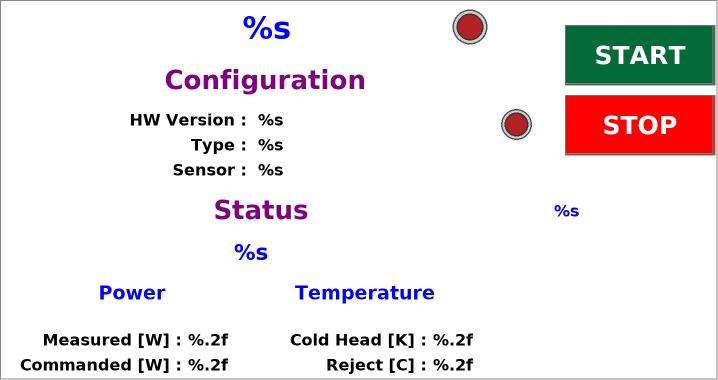
VISUALIZATION GUI_TEMPLATE_CRYOTELGT  // 718x380
VAR_IN_OUT
	m_Instance:	FB_CRYO_CRYOTELGT;
	m_bEnable:	BOOL;	// Flag to start/stop the cooler
END_VAR
    Rectangle (159,65 213x30), "Configuration"
    Rectangle (186,195 150x30), "Status"
    Rectangle (25,325 160x30), "Measured [W] :", tooltip "'P' command: Measured Power"
    Rectangle (185,325 70x30), "%.2f", text variable: m_Instance.stat.lrPowerMeasured
    Rectangle (152,10 230x36), "%s", text variable: m_Instance.in_sName
    Rectangle (255,155 110x30), "%s", text variable: m_Instance.stat.sSensor
    Rectangle (255,105 100x30), "%s", text variable: m_Instance.stat.sVersion
    Rectangle (255,130 100x30), "%s", text variable: m_Instance.stat.sMode
    Button (565,25 150x60), "START"
        OnMouseClick: execute { m_bEnable := TRUE; }
    Button (565,95 150x60), "STOP"
        OnMouseClick: execute { m_bEnable := FALSE; }
    Lamp1 (499,107 35x35), tooltip "If ON, there is a communication problem with the Cooler.", variable: m_Instance.bCommProblem, style: Lamp-Lamp1-Red
    Rectangle (36,235 431x35), "%s", tooltip "'COOLER' command: Cooler Control Mode: OFF or POWER", text variable: m_Instance.stat.sCtrlMode
    Rectangle (105,105 145x30), "HW Version :", tooltip "'VERSION' command: Current controller code version"
    Rectangle (105,130 145x30), "Type :", tooltip "'MODE' command: Cryocooler type, e.g. GT"
    Rectangle (105,155 145x30), "Sensor :", tooltip "'SENSOR' command: Configured temp. sensor type, e.g. 'PT-100'"
    Rectangle (57,278 150x30), "Power"
    Rectangle (290,278 150x30), "Temperature"
    Rectangle (25,350 160x30), "Commanded [W] :", tooltip "'PWOUT' command: Commanded power"
    Rectangle (185,350 70x30), "%.2f", text variable: m_Instance.stat.lrPowerCommanded
    Rectangle (285,325 145x30), "Cold Head [K] :", tooltip "'TC' command: Cold Head temperature"
    Rectangle (430,325 70x30), "%.2f", text variable: m_Instance.stat.lrTempColdHead
    Rectangle (285,350 145x30), "Reject [C] :", tooltip "'TEMP RJ' command: Reject Temperature"
    Rectangle (430,350 70x30), "%.2f", text variable: m_Instance.stat.lrTempReject
    Rectangle (416,196 302x30), "%s", tooltip "Cooler State", text variable: m_Instance.stat.sDevState
    Lamp1 (450,7 40x40), tooltip "If ON, Cooler is simulated.", variable: m_Instance.stat.bSimulation, invisible if: m_Instance.in_bSimulation = FALSE, style: Lamp-Lamp1-Red
END_VISUALIZATION

// ---- VISUs/Templates/GUI_TEMPLATE_CRYO_CPA.TcVIS
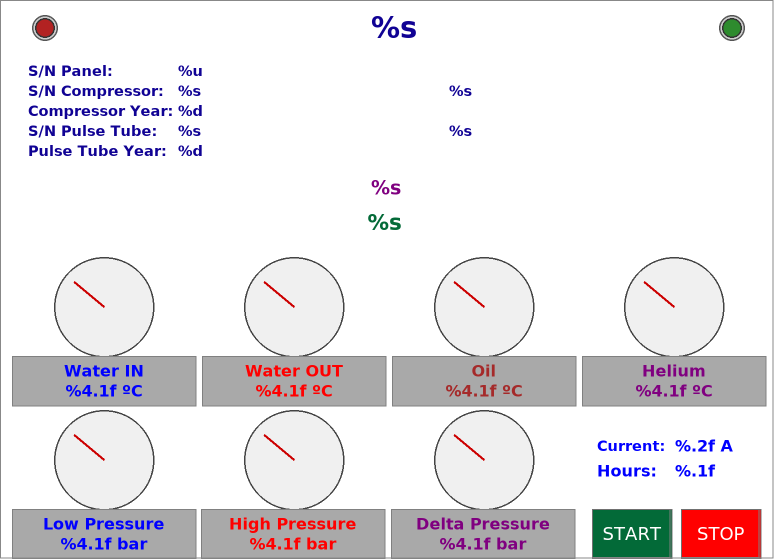
VISUALIZATION GUI_TEMPLATE_CRYO_CPA  // 774x559
VAR_IN_OUT
	m_Instance:	FB_CRYO_CPA;
END_VAR
    Rectangle (80,10 629x35), "%s", text variable: m_Instance.stat.sModelNumber
    Rectangle (10,207 750x30), "%s", text variable: m_Instance.stat.sError, invisible if: (m_Instance.stat.nStatusCode<>2)
    Meter180 (4,410 200x100), value: m_Instance.stat.lrLowPressure, style: Meter-Meter180-Gray, scale format: %.0f, scale 0..30
    Rectangle (12,509 184x50), "Low Pressure %4.1f bar", text variable: m_Instance.stat.lrLowPressure
    Meter180 (194,410 200x100), value: m_Instance.stat.lrHighPressure, style: Meter-Meter180-Gray, scale format: %.0f, scale 0..30
    Rectangle (201,509 184x50), "High Pressure %4.1f bar", text variable: m_Instance.stat.lrHighPressure
    Lamp1 (717,13 30x30), tooltip "If ON, compressor is running", variable: m_Instance.stat.bSystemOn, style: Lamp-Lamp1-Green
    Rectangle (10,208 750x30), "%s", text variable: m_Instance.stat.sAlarm, invisible if: (m_Instance.stat.nStatusCode<>1)
    Rectangle (231,206 308x33), "%s", text variable: m_Instance.stat.sStatusOK, invisible if: (m_Instance.stat.nStatusCode<>0 or m_Instance.stat.nOperatingState <>3)
    Meter180 (4,257 200x100), value: m_Instance.stat.lrCoolantInTemp, style: Meter-Meter180-Gray, scale format: %.0f, scale 0..60
    Rectangle (12,356 184x50), "Water IN %4.1f ºC", text variable: m_Instance.stat.lrCoolantInTemp
    Meter180 (194,257 200x100), value: m_Instance.stat.lrCoolantOutTemp, style: Meter-Meter180-Gray, scale format: %.0f, scale 0..60
    Rectangle (202,356 184x50), "Water OUT %4.1f ºC", text variable: m_Instance.stat.lrCoolantOutTemp
    Meter180 (384,257 200x100), value: m_Instance.stat.lrOilTemp, style: Meter-Meter180-Gray, scale format: %.0f, scale 0..60
    Rectangle (392,356 184x50), "Oil %4.1f ºC", text variable: m_Instance.stat.lrOilTemp
    Meter180 (574,257 200x100), value: m_Instance.stat.lrHeliumTemp, style: Meter-Meter180-Gray, scale format: %.0f, scale 0..100
    Rectangle (582,356 184x50), "Helium %4.1f ºC", text variable: m_Instance.stat.lrHeliumTemp
    Rectangle (672,431 95x30), "%.2f A", text variable: m_Instance.stat.lrMotorCurrent
    Rectangle (672,456 95x30), "%.1f", text variable: m_Instance.stat.lrHoursOfOperation
    Rectangle (140,173 493x30), "%s", tooltip "Operational State", text variable: m_Instance.stat.sOperatingState
    Rectangle (175,60 231x22), "%u", text variable: m_Instance.stat.nPanelSerialNumber
    Rectangle (175,80 270x22), "%s", text variable: m_Instance.in_sSN_Compressor
    Rectangle (175,120 270x22), "%s", text variable: m_Instance.in_sSN_PulseTube
    Label (25,60 145x22), "S/N Panel:"
    Label (25,80 145x22), "S/N Compressor:"
    Label (25,120 145x22), "S/N Pulse Tube:"
    Rectangle (594,431 75x30), "Current:"
    Rectangle (594,456 75x30), "Hours:"
    Meter180 (384,410 200x100), value: m_Instance.stat.lrDeltaPressureAverage, style: Meter-Meter180-Gray, scale format: %.0f, scale 0..30
    Rectangle (391,509 184x50), "Delta Pressure %4.1f bar", text variable: m_Instance.stat.lrDeltaPressureAverage
    Label (25,140 145x22), "Pulse Tube Year:"
    Rectangle (175,140 90x22), "%d", text variable: m_Instance.in_nYear_PulseTube
    Label (25,100 145x22), "Compressor Year:"
    Rectangle (175,100 90x22), "%d", text variable: m_Instance.in_nYear_Compressor
    Rectangle (446,80 270x22), "%s", text variable: m_Instance.stat.sServiceDue_Compressor, invisible if: m_Instance.stat.bServiceDue_Compressor=FALSE
        p55702900: m_Instance.stat.wColour_Compressor
    Rectangle (446,120 270x22), "%s", text variable: m_Instance.stat.sServiceDue_PulseTube, invisible if: m_Instance.stat.bServiceDue_PulseTube=FALSE
        p55702900: m_Instance.stat.wColour_PulseTube
    Button (592,509 80x50), "START", input disabled if: m_Instance.stat.bSystemOn
        OnMouseClick: execute { m_Instance.ctrl.nDevCommand := E_CRYO_CPA_CMDS.START; m_Instance.ctrl.bExecute := TRUE; }
    Button (681,509 80x50), "STOP", input disabled if: NOT m_Instance.stat.bSystemOn
        OnMouseClick: execute { m_Instance.ctrl.nDevCommand := E_CRYO_CPA_CMDS.STOP; m_Instance.ctrl.bExecute := TRUE; }
    Lamp1 (30,13 30x30), tooltip "If ON, compressor is simulated", variable: m_Instance.stat.bSimulation, invisible if: m_Instance.stat.bSimulation=false, style: Lamp-Lamp1-Red
END_VISUALIZATION

// ---- VISUs/Templates/GUI_TEMPLATE_CRYO_EVAC_BASE.TcVIS
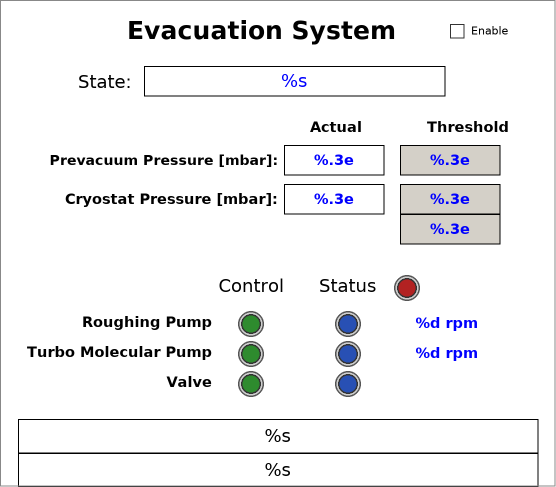
VISUALIZATION GUI_TEMPLATE_CRYO_EVAC_BASE  // 556x487
VAR_IN_OUT
	m_Instance:	FB_CRYO_EVAC_BASE;
	m_bEnable:	BOOL;
END_VAR
    Rectangle (144,66 301x30), "%s", text variable: m_Instance.stat.sState
    Lamp1 (236,309 30x30), variable: m_Instance.ctrl.bEnable_RP, style: Lamp-Lamp1-Green
    Rectangle (15,307 200x30), "Roughing Pump"
    Lamp1 (236,339 30x30), variable: m_Instance.ctrl.bEnable_TP, style: Lamp-Lamp1-Green
    Rectangle (15,337 200x30), "Turbo Molecular Pump"
    Lamp1 (236,369 30x30), variable: m_Instance.ctrl.bEnable_Valve, style: Lamp-Lamp1-Green
    Rectangle (15,367 200x30), "Valve"
    Rectangle (18,419 520x34), "%s", tooltip "Error description", text variable: m_Instance.stat.sErrorText
    Checkbox (448,16 108x30), "Enable", variable: m_bEnable
    Rectangle (56,67 84x30), "State:"
    Rectangle (299,271 98x30), "Status"
    Rectangle (284,145 100x30), "%.3e", tooltip "Prevacuum pressure [mbar]", text variable: m_Instance.prevac.stat.lrPressure
    Rectangle (400,145 100x30), "%.3e", tooltip "Prevacuum pressure threshold [mbar]", text variable: m_Instance.cfg.lrThld_Prevac
    Rectangle (284,184 100x30), "%.3e", tooltip "Cryo pressure [mbar]", text variable: m_Instance.in_lrCryoPressure
    Rectangle (400,184 100x30), "%.3e", tooltip "Pressure threshold for safe start of Turbo Pump [mbar]", text variable: m_Instance.cfg.lrThld_TP_SafeStartPressure
    Rectangle (400,214 100x30), "%.3e", tooltip "Pressure threshold for safe opening of the pre-vacuum valve [mbar]", text variable: m_Instance.cfg.lrThld_Valve_SafeOpenPressure
    Rectangle (51,145 230x30), "Prevacuum Pressure [mbar]:"
    Rectangle (51,184 230x30), "Cryostat Pressure [mbar]:"
    Rectangle (307,112 232x30), "Actual Threshold"
    Lamp1 (333,309 30x30), tooltip "If ON, Pump is Running", variable: m_Instance.stat.bRootPumpON, style: Lamp-Lamp1-Blue
    Lamp1 (333,339 30x30), tooltip "If ON, Pump is Running", variable: m_Instance.stat.bTurboPumpON, style: Lamp-Lamp1-Blue
    Lamp1 (333,369 30x30), tooltip "If ON, Insulation Valve is OPEN", variable: m_Instance.valve.stat.bActON, style: Lamp-Lamp1-Blue
    Rectangle (381,308 100x30), "%d rpm", tooltip "Roughing Pump Speed [rpm]", text variable: m_Instance.rpRef.statBaseRef.nPumpSpeed
    Rectangle (381,338 100x30), "%d rpm", tooltip "Turbo Pump Speed [rpm]", text variable: m_Instance.tp.stat.nPumpSpeed
    Rectangle (92,13 339x34), "Evacuation System"
    Rectangle (195,271 113x30), "Control"
    Rectangle (18,453 520x34), "%s", tooltip "Evacuation System Status", text variable: m_Instance.stat.sStatus
    Lamp1 (392,273 30x30), tooltip "If ON, there was an error", variable: m_Instance.stat.bError, style: Lamp-Lamp1-Red
END_VISUALIZATION

// ---- VISUs/Templates/GUI_TEMPLATE_ECODRY_V01.TcVIS
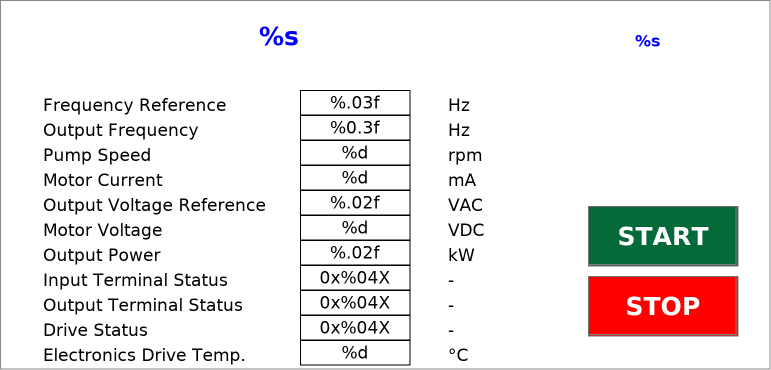
VISUALIZATION GUI_TEMPLATE_ECODRY_V01  // 771x370
VAR_IN_OUT
	m_Instance:	FB_CRYO_PUMP_ECODRY;
	m_bEnable:	BOOL;	// Flag to start/stop the pump
END_VAR
    Rectangle (300,90 110x25), "%.03f", text variable: m_Instance.stat.lrFreqRef
    Rectangle (300,115 110x25), "%0.3f", text variable: m_Instance.stat.lrOutFreq
    Rectangle (300,165 110x25), "%d", text variable: m_Instance.stat.nMotorCurr
    Rectangle (300,190 110x25), "%.02f", text variable: m_Instance.stat.lrOutVoltRef
    Label (40,90 245x30), "Frequency Reference"
    Label (40,115 245x30), "Output Frequency"
    Label (40,165 245x30), "Motor Current"
    Label (40,190 245x30), "Output Voltage Reference"
    Rectangle (300,215 110x25), "%d", text variable: m_Instance.stat.nMotorVolt
    Rectangle (300,240 110x25), "%.02f", text variable: m_Instance.stat.lrOutPower
    Rectangle (300,265 110x25), "0x%04X"
    Rectangle (300,290 110x25), "0x%04X"
    Label (40,215 245x30), "Motor Voltage"
    Label (40,240 245x30), "Output Power"
    Label (40,265 245x30), "Input Terminal Status"
    Label (40,290 245x30), "Output Terminal Status"
    Rectangle (300,315 110x25), "0x%04X"
    Rectangle (300,340 110x25), "%d", text variable: m_Instance.stat.nElecTemp
    Label (40,315 245x30), "Drive Status"
    Label (40,340 245x30), "Electronics Drive Temp."
    Label (445,90 59x30), "Hz"
    Label (445,115 59x30), "Hz"
    Label (445,165 59x30), "mA"
    Label (445,190 59x30), "VAC"
    Label (445,215 59x30), "VDC"
    Label (445,240 59x30), "kW"
    Label (445,265 59x30), "-"
    Label (445,290 59x30), "-"
    Label (445,315 59x30), "-"
    Label (445,340 59x30), "°C"
    Rectangle (164,21 230x30), "%s", text variable: m_Instance.in_sName
    Button (588,206 150x60), "START"
        OnMouseClick: execute { m_bEnable := TRUE; }
    Button (588,276 150x60), "STOP"
        OnMouseClick: execute { m_bEnable := FALSE; }
    Rectangle (525,26 246x30), "%s", tooltip "Control Mode", text variable: m_Instance.stat.sPumpState
    Rectangle (300,140 110x25), "%d", text variable: m_Instance.stat.nPumpSpeed
    Label (40,140 245x30), "Pump Speed"
    Label (445,140 59x30), "rpm"
END_VISUALIZATION

// ---- VISUs/Templates/GUI_TEMPLATE_HIPACE_30.TcVIS
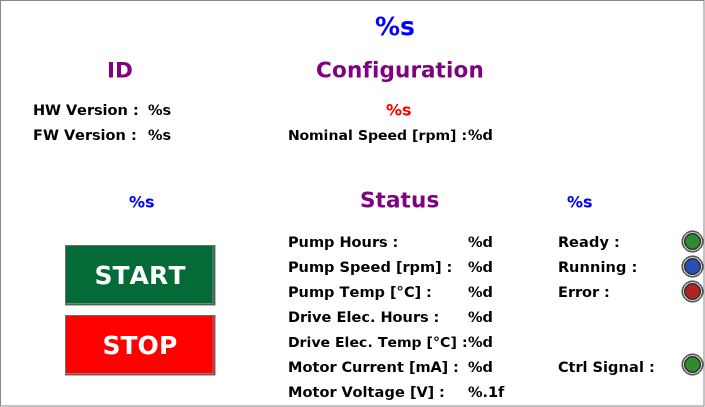
VISUALIZATION GUI_TEMPLATE_HIPACE_30  // 705x407
VAR_IN_OUT
	m_Instance:	FB_CRYO_PUMP_HIPACE30;
	m_bEnable:	BOOL;	// Flag to start/stop the pump
END_VAR
    Rectangle (45,55 150x30), "ID"
    Rectangle (310,55 180x30), "Configuration"
    Rectangle (325,185 150x30), "Status"
    Lamp1 (680,229 25x25), tooltip "OK for Process, i.e. speed ≥ nominal speed", variable: m_Instance.stat.bReady, style: Lamp-Lamp1-Green
    Lamp1 (680,254 25x25), tooltip "pump speed > 0 rpm", variable: m_Instance.stat.bMoving, style: Lamp-Lamp1-Blue
    Lamp1 (680,279 25x25), tooltip "presence of a warning", variable: m_Instance.stat.bFailure, style: Lamp-Lamp1-Red
    Rectangle (555,227 110x30), "Ready :"
    Rectangle (555,252 110x30), "Running :"
    Rectangle (555,277 110x30), "Error :"
    Rectangle (285,120 180x30), "Nominal Speed [rpm] :"
    Rectangle (285,227 180x30), "Pump Hours :"
    Rectangle (285,302 180x30), "Drive Elec. Hours :"
    Rectangle (465,120 70x30), "%d", text variable: m_Instance.stat.nNominalSpeed
    Rectangle (465,227 70x30), "%d", text variable: m_Instance.stat.nPumpHours
    Rectangle (465,302 70x30), "%d", text variable: m_Instance.stat.nElecHours
    Rectangle (285,252 180x30), "Pump Speed [rpm] :"
    Rectangle (465,252 70x30), "%d", text variable: m_Instance.stat.nPumpSpeed
    Rectangle (285,327 180x30), "Drive Elec. Temp [°C] :", text variable: m_Instance.stat.nElecTemp
    Rectangle (465,327 70x30), "%d", text variable: m_Instance.stat.nElecTemp
    Rectangle (285,277 180x30), "Pump Temp [°C] :"
    Rectangle (465,277 70x30), "%d", text variable: m_Instance.stat.nPumpTemp
    Rectangle (285,352 180x30), "Motor Current [mA] :", text variable: m_Instance.stat.nMotorCurr
    Rectangle (465,352 70x30), "%d", text variable: m_Instance.stat.nMotorCurr
    Rectangle (285,377 180x30), "Motor Voltage [V] :", text variable: m_Instance.stat.nMotorVolt
    Rectangle (465,377 70x30), "%.1f", text variable: m_Instance.stat.lrMotorVolt
    Rectangle (280,11 230x30), "%s", text variable: m_Instance.in_sName
    Rectangle (289,95 220x30), "%s", tooltip "Control Mode", text variable: m_Instance.stat.sCtrlMode
    Rectangle (145,95 130x30), "%s", tooltip "HW Version", text variable: m_Instance.stat.sHwVersion
    Rectangle (145,120 130x30), "%s", tooltip "FW Version", text variable: m_Instance.stat.sFwVersion
    Button (65,245 150x60), "START"
        OnMouseClick: execute { m_bEnable := TRUE; }
    Button (65,315 150x60), "STOP"
        OnMouseClick: execute { m_bEnable := FALSE; }
    Lamp1 (680,352 25x25), tooltip "If ON, control output signal is active.", variable: m_Instance.q_bStart, style: Lamp-Lamp1-Green
    Rectangle (555,352 110x30), "Ctrl Signal :"
    Rectangle (457,187 246x30), "%s", tooltip "Pump State", text variable: m_Instance.stat.sPumpState
    Rectangle (92,187 100x30), "%s", tooltip "Error Status", text variable: m_Instance.stat.sFailureCode
    Rectangle (30,95 110x30), "HW Version :"
    Rectangle (30,120 110x30), "FW Version :"
END_VISUALIZATION

// ---- VISUs/Templates/GUI_TEMPLATE_MVP030.TcVIS
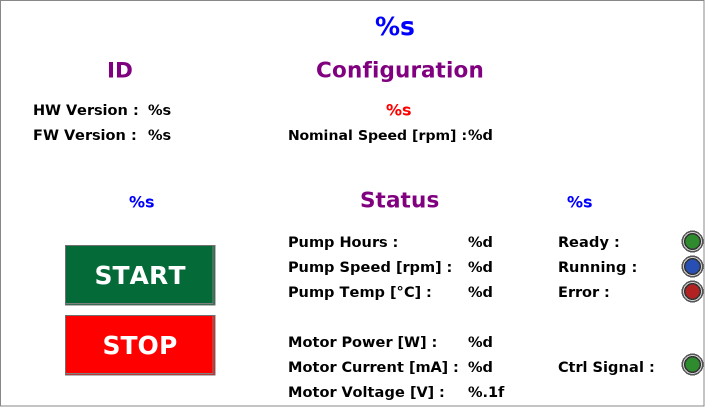
VISUALIZATION GUI_TEMPLATE_MVP030  // 705x407
VAR_IN_OUT
	m_Instance:	FB_CRYO_PUMP_MVP030;
	m_bEnable:	BOOL;	// Flag to start/stop the pump
END_VAR
    Rectangle (45,55 150x30), "ID"
    Rectangle (310,55 180x30), "Configuration"
    Rectangle (325,185 150x30), "Status"
    Lamp1 (680,229 25x25), tooltip "OK for Process, i.e. speed ≥ nominal speed", variable: m_Instance.stat.bReady, style: Lamp-Lamp1-Green
    Lamp1 (680,254 25x25), tooltip "pump speed > 0 rpm", variable: m_Instance.stat.bMoving, style: Lamp-Lamp1-Blue
    Lamp1 (680,279 25x25), tooltip "presence of a warning", variable: m_Instance.stat.bFailure, style: Lamp-Lamp1-Red
    Rectangle (555,227 110x30), "Ready :"
    Rectangle (555,252 110x30), "Running :"
    Rectangle (555,277 110x30), "Error :"
    Rectangle (285,120 180x30), "Nominal Speed [rpm] :"
    Rectangle (285,227 180x30), "Pump Hours :"
    Rectangle (465,120 70x30), "%d", text variable: m_Instance.stat.nNominalSpeed
    Rectangle (465,227 70x30), "%d", text variable: m_Instance.stat.nPumpHours
    Rectangle (285,252 180x30), "Pump Speed [rpm] :"
    Rectangle (465,252 70x30), "%d", text variable: m_Instance.stat.nPumpSpeed
    Rectangle (285,277 180x30), "Pump Temp [°C] :"
    Rectangle (465,277 70x30), "%d", text variable: m_Instance.stat.nPumpTemp
    Rectangle (285,352 180x30), "Motor Current [mA] :"
    Rectangle (465,352 70x30), "%d", text variable: m_Instance.stat.nMotorCurr
    Rectangle (285,377 180x30), "Motor Voltage [V] :"
    Rectangle (465,377 70x30), "%.1f", text variable: m_Instance.stat.lrMotorVolt
    Rectangle (280,11 230x30), "%s", text variable: m_Instance.in_sName
    Rectangle (289,95 220x30), "%s", tooltip "Control Mode", text variable: m_Instance.stat.sCtrlMode
    Rectangle (145,95 130x30), "%s", tooltip "HW Version", text variable: m_Instance.stat.sHwVersion
    Rectangle (145,120 130x30), "%s", tooltip "FW Version", text variable: m_Instance.stat.sFwVersion
    Button (65,245 150x60), "START"
        OnMouseClick: execute { m_bEnable := TRUE; }
    Button (65,315 150x60), "STOP"
        OnMouseClick: execute { m_bEnable := FALSE; }
    Lamp1 (680,352 25x25), tooltip "If ON, control output signal is active.", variable: m_Instance.q_bStart, style: Lamp-Lamp1-Green
    Rectangle (555,352 110x30), "Ctrl Signal :"
    Rectangle (457,187 246x30), "%s", tooltip "Pump State", text variable: m_Instance.stat.sPumpState
    Rectangle (92,187 100x30), "%s", tooltip "Error Status", text variable: m_Instance.stat.sFailureCode
    Rectangle (285,327 180x30), "Motor Power [W] :"
    Rectangle (465,327 70x30), "%d", text variable: m_Instance.stat.nElecPower
    Rectangle (30,95 110x30), "HW Version :"
    Rectangle (30,120 110x30), "FW Version :"
END_VISUALIZATION

// ---- VISUs/Templates/GUI_TEMPLATE_SBG232.TcVIS
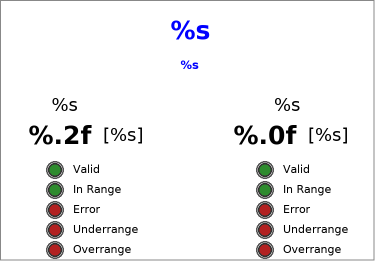
VISUALIZATION GUI_TEMPLATE_SBG232  // 375x261
VAR_IN_OUT
	m_Instance:	FB_CRYO_SBG232;
END_VAR
    Rectangle (41,10 299x40), "%s", tooltip "Sensor Name", text variable: m_Instance.stat.sName
    Rectangle (20,120 80x30), "%.2f", text variable: m_Instance.stat.flow.lrValue
    Rectangle (30,90 70x30), "%s", text variable: m_Instance.stat.flow.sType
    Rectangle (100,120 70x30), "[%s]", text variable: m_Instance.stat.flow.sUnits
    Rectangle (225,120 80x30), "%.0f", text variable: m_Instance.stat.temp.lrValue
    Rectangle (220,90 135x30), "%s", text variable: m_Instance.stat.temp.sType
    Rectangle (305,120 70x30), "[%s]", text variable: m_Instance.stat.temp.sUnits
    Lamp1 (45,160 20x20), tooltip "If ON, reading is valid.", variable: m_Instance.stat.flow.bValid, style: Lamp-Lamp1-Green
    Lamp1 (45,180 20x20), tooltip "If ON, reading is in expected range.", variable: m_Instance.stat.flow.bInRange, style: Lamp-Lamp1-Green
    Rectangle (5,50 370x30), "%s", tooltip "Sensor Status", text variable: m_Instance.stat.sStatus
    Lamp1 (45,220 20x20), tooltip "If ON, reading is in underrange.", variable: m_Instance.stat.flow.bUnderrange, style: Lamp-Lamp1-Red
    Lamp1 (45,240 20x20), tooltip "If ON, reading is in overrange.", variable: m_Instance.stat.flow.bOverrange, style: Lamp-Lamp1-Red
    Lamp1 (45,200 20x20), tooltip "If ON, reading is in error.", variable: m_Instance.stat.flow.bError, style: Lamp-Lamp1-Red
    Label (70,158 87x23), "Valid"
    Label (70,178 87x23), "In Range"
    Label (70,198 87x23), "Error"
    Label (70,218 87x23), "Underrange"
    Label (70,238 87x23), "Overrange"
    Lamp1 (255,160 20x20), tooltip "If ON, reading is valid.", variable: m_Instance.stat.temp.bValid, style: Lamp-Lamp1-Green
    Lamp1 (255,180 20x20), tooltip "If ON, reading is in expected range.", variable: m_Instance.stat.temp.bInRange, style: Lamp-Lamp1-Green
    Lamp1 (255,220 20x20), tooltip "If ON, reading is in underrange.", variable: m_Instance.stat.temp.bUnderrange, style: Lamp-Lamp1-Red
    Lamp1 (255,240 20x20), tooltip "If ON, reading is in overrange.", variable: m_Instance.stat.temp.bOverrange, style: Lamp-Lamp1-Red
    Lamp1 (255,200 20x20), tooltip "If ON, reading is in error.", variable: m_Instance.stat.temp.bError, style: Lamp-Lamp1-Red
    Label (280,158 87x23), "Valid"
    Label (280,178 87x23), "In Range"
    Label (280,198 87x23), "Error"
    Label (280,218 87x23), "Underrange"
    Label (280,238 87x23), "Overrange"
END_VISUALIZATION

// ---- VISUs/Templates/GUI_TEMPLATE_TEMP_OVERRIDE.TcVIS
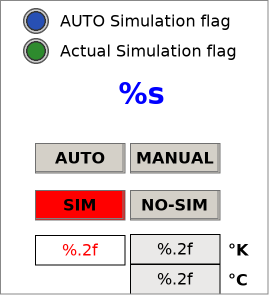
VISUALIZATION GUI_TEMPLATE_TEMP_OVERRIDE  // 269x295
VAR_IN_OUT
	m_Cmd:		FB_CRYO_CMD_OVERRIDE;
	m_Temp:		FB_CRYO_TEMPERATURE;
END_VAR
    Button (35,190 90x30), "SIM", tooltip "Activate Simulation", colour toggle: (m_Cmd.bPermitOn AND NOT m_Cmd.bAutoMode) OR m_Cmd.bEngMode, input disabled if: m_Cmd.bDisableBtnOn
        OnMouseClick: execute { m_Cmd.bManualCmd := TRUE; }
    Lamp1 (21,36 30x30), tooltip "Actual Simulation flag going out", variable: m_Cmd.out_bEnable, style: Lamp-Lamp1-Green
    Rectangle (57,36 200x30), "Actual Simulation flag", tooltip "Actual Simulation flag set the user"
    Button (35,143 90x30), "AUTO", tooltip "Switch to AUTO Mode", colour toggle: m_Cmd.bAutoMode, input disabled if: m_Cmd.bAutoMode OR m_Cmd.bEngMode
        OnMouseClick: execute { m_Cmd.bAutoMode := TRUE; }
    Button (130,143 90x30), "MANUAL", tooltip "Switch to MANUAL Mode", colour toggle: NOT m_Cmd.bAutoMode, input disabled if: NOT m_Cmd.bAutoMode AND NOT m_Cmd.bEngMode
        OnMouseClick: execute { m_Cmd.bAutoMode := FALSE; }
    Button (130,190 90x30), "NO-SIM", tooltip "Deactivate Simulation", colour toggle: (m_Cmd.bPermitOff AND NOT m_Cmd.bAutoMode) OR m_Cmd.bEngMode, input disabled if: m_Cmd.bDisableBtnOff
        OnMouseClick: execute { m_Cmd.bManualCmd := FALSE; }
    Lamp1 (21,6 30x30), tooltip "Simulation flag coming from the Control System", variable: m_Cmd.in_bEnable, style: Lamp-Lamp1-Blue
    Rectangle (57,6 200x30), "AUTO Simulation flag", tooltip "AUTO Simulation flag set by the system"
    Rectangle (67,73 150x41), "%s", text variable: m_Cmd.out_sMode
    Rectangle (35,235 90x30), "%.2f", tooltip "Simulated value [K] when simulation is active.", text variable: m_Temp.stat.lrSimTempK, input disabled if: m_Cmd.bDisableBtnOn OR NOT m_Cmd.out_bEnable
        OnMouseClick: write the text variable via Default
    Rectangle (130,234 90x30), "%.2f", tooltip "Value used by the system [K]", text variable: m_Temp.stat.lrTempK
    Label (225,235 44x30), "°K"
    Rectangle (130,264 90x30), "%.2f", tooltip "Value used by the system [C]", text variable: m_Temp.stat.lrTempC
    Label (225,265 44x30), "°C"
END_VISUALIZATION

// ---- VISUs/Templates/GUI_TEMPLATE_PRESS_OVERRIDE.TcVIS
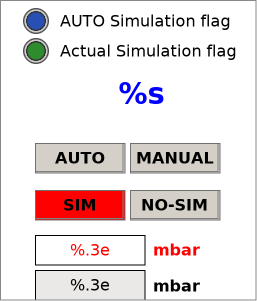
VISUALIZATION GUI_TEMPLATE_PRESS_OVERRIDE  // 257x301
VAR_IN_OUT
	m_Cmd:		FB_CRYO_CMD_OVERRIDE;
	m_Press:	FB_CRYO_PRESSURE_VOTE;
END_VAR
    Button (35,190 90x30), "SIM", tooltip "Activate Simulation", colour toggle: (m_Cmd.bPermitOn AND NOT m_Cmd.bAutoMode) OR m_Cmd.bEngMode, input disabled if: m_Cmd.bDisableBtnOn
        OnMouseClick: execute { m_Cmd.bManualCmd := TRUE; }
    Lamp1 (21,36 30x30), tooltip "Actual Simulation flag going out", variable: m_Cmd.out_bEnable, style: Lamp-Lamp1-Green
    Rectangle (57,36 200x30), "Actual Simulation flag", tooltip "Actual Simulation flag set the user"
    Button (35,143 90x30), "AUTO", tooltip "Switch to AUTO Mode", colour toggle: m_Cmd.bAutoMode, input disabled if: m_Cmd.bAutoMode OR m_Cmd.bEngMode
        OnMouseClick: execute { m_Cmd.bAutoMode := TRUE; }
    Button (130,143 90x30), "MANUAL", tooltip "Switch to MANUAL Mode", colour toggle: NOT m_Cmd.bAutoMode, input disabled if: NOT m_Cmd.bAutoMode AND NOT m_Cmd.bEngMode
        OnMouseClick: execute { m_Cmd.bAutoMode := FALSE; }
    Button (130,190 90x30), "NO-SIM", tooltip "Deactivate Simulation", colour toggle: (m_Cmd.bPermitOff AND NOT m_Cmd.bAutoMode) OR m_Cmd.bEngMode, input disabled if: m_Cmd.bDisableBtnOff
        OnMouseClick: execute { m_Cmd.bManualCmd := FALSE; }
    Lamp1 (21,6 30x30), tooltip "Simulation flag coming from the Control System", variable: m_Cmd.in_bEnable, style: Lamp-Lamp1-Blue
    Rectangle (57,6 200x30), "AUTO Simulation flag", tooltip "AUTO Simulation flag set by the system"
    Rectangle (67,73 150x41), "%s", text variable: m_Cmd.out_sMode
    Rectangle (35,235 110x30), "%.3e", tooltip "Simulated value [mbar] when simulation is active.", text variable: m_Press.stat.lrSimPressure, input disabled if: m_Cmd.bDisableBtnOn OR NOT m_Cmd.out_bEnable
        OnMouseClick: write the text variable via Default
    Rectangle (35,270 110x30), "%.3e", tooltip "Value used by the system [mbar]", text variable: m_Press.stat.lrPressure
    Label (150,271 50x30), "mbar"
    Label (150,235 50x30), "mbar"
END_VISUALIZATION
